// TIA Portal V20 export
// export: Created 2025-12-01T14:57:26.8993515Z, ExportSetting None, DisplayName Totally Integrated Automation Portal, DisplayVersion V20 Update 3, DisplayName TIA Portal Openness, DisplayVersion V20 Update 3, DisplayName TIA Portal Version Control Interface, DisplayVersion V20 Update 3, DisplayName STEP 7 Professional, DisplayVersion V20 Update 3, DisplayName STEP 7 Safety, DisplayVersion V20 Update 2, DisplayName WinCC Basic/Comfort/Advanced, DisplayVersion V20 Update 3, DisplayName WinCC Professional, DisplayVersion V20 Update 3, DisplayName WinCC Unified, DisplayVersion V20 Update 3
FUNCTION "FC606_EventosEnv_Quimarox" : Void   // FC606, LAD
{ S7_Optimized_Access := 'FALSE' }
// stored: AutoNumber false, SetENOAutomatically false
   VAR_INPUT
      NumQuimarox : UInt;
   END_VAR
   VAR_TEMP
      P_Eventos : DWord;
      DBEventos : Word;
      NumDBEventos : UInt;
      MaxBytes : UInt;
      Valor : UDInt;
      NumBytes : UInt;
      Offset : UInt;
      NumVagon : UInt;
      MesaAsociada : UInt;
      MaxNumVagones : UInt;
      EventoAGenerar : UInt;
      Cero : Byte;
      ReturnValor : Int;
      Reserva_Elemento : UInt;
      Reserva_Activa : Bool;
   END_VAR
BEGIN

NETWORK
TITLE = Inicializar
///////////////////////////////////////////////////////////////////////////////////////////
///////////////////////////////////////////////////////////////////////////////////////////
///////////////////////////////////////////////////////////////////////////////////////////
/// Datos del quimarox (Vagon = Peine)
/// ---  Mesa Asociada al Quimarox
/// ---  Maximo Numero de Vagones en el Quimarox

      L     "DB600_ConfigQuimarox".Quimarox[#NumQuimarox].datos_config.Numero_MesaAsociada;
      T     #MesaAsociada;  // Mesa Asociada
      L     "DB600_ConfigQuimarox".Quimarox[#NumQuimarox].datos_config.Numero_vagones;
      T     #MaxNumVagones;  // Numero Maximo De Vagones



NETWORK
TITLE = Comprobacion de Existencia de Eventos en los Vagones
///////////////////////////////////////////////////////////////////////////////////////////
///////////////////////////////////////////////////////////////////////////////////////////
///////////////////////////////////////////////////////////////////////////////////////////
/// Inicio del Recorrido de Vagones Existentes en el Quimarox

      L     1;
      T     #NumVagon;


///////////////////////////////////////////////////////////////////////////////////////////
BucleVagonesQuimarox:NOP   0;
      L     "DB601_PeinesQuimarox".Quimarox[#NumQuimarox].vagon[#NumVagon].EventoAGenerar;
      T     #EventoAGenerar;  // Leer Numero de Evento A Generar

      L     #EventoAGenerar;  // Hay Evento a Generar ?
      L     0;
      <>I;
      JC    GenerarEvento;
      JU    Siguiente_VagonQuimarox;  // Siguiente Vagon


///////////////////////////////////////////////////////////////////////////////////////////
// Continuar Recorriendo los Vagones del Quimarox
Siguiente_VagonQuimarox:NOP   0;
      L     #NumVagon;  // Siguiente Numero de Vagon
      L     1;  // +1
      +I;
      T     #NumVagon;

      L     #NumVagon;  // Es final de los Vagones del Quimarox ?
      L     #MaxNumVagones;
      >I;
      JC    FinalBucleVagonesQuimarox;
      JU    BucleVagonesQuimarox;


///////////////////////////////////////////////////////////////////////////////////////////
///////////////////////////////////////////////////////////////////////////////////////////
///////////////////////////////////////////////////////////////////////////////////////////
/// Final del Recorrido de Vagones existentes en el Quimarox
FinalBucleVagonesQuimarox:NOP   0;
      JU    Final_Funcion;  // Final de la Funcion



NETWORK
TITLE = Inicio de la Generacion del Evento
GenerarEvento:NOP   0;

///////////////////////////////////////////////////////////////////////////////////////////
///////////////////////////////////////////////////////////////////////////////////////////
///////////////////////////////////////////////////////////////////////////////////////////
/// Recoger los Datos del DB a Escribir los Eventos

      L     "JDT1_NDB_EventosEmi";  // Datos del JDT01
      T     #DBEventos;
      T     #NumDBEventos;
      L     "JDT1_MaxBytes";
      T     #MaxBytes;

      SET;
      AN    "DB850_DefinicionMesas".Mesa[#MesaAsociada].ConfigMesa.MesaDeJDT02;
      JC    NoEs_MesaJDT02;  // Es de JDT02 ?


      L     "JDT2_NDB_EventosEmi";  // Datos del JDT02
      T     #DBEventos;
      T     #NumDBEventos;
      L     "JDT2_MaxBytes";
      T     #MaxBytes;

///////////////////////////////////////////////////////////////////////////////////////////
NoEs_MesaJDT02:NOP   0;




NETWORK
TITLE = ---
///////////////////////////////////////////////////////////////////////////////////////////
///////////////////////////////////////////////////////////////////////////////////////////
///////////////////////////////////////////////////////////////////////////////////////////
/// Comprobacion si hay sitio para Formatear el Evento

      L     0;
      T     #NumBytes;  // Inicializo el numero de Bytes
      T     #P_Eventos;  // Inicializo el puntero de Eventos Generados

Inicio_BusquedaFinalEventos:NOP   0;
      OPN   DB [#DBEventos];  // Calcula el tamaño de bytes que hay en el DB
      L     DBB [#P_Eventos];
      L     0;
      ==I;
      JC    Fin_BusquedaFinalEventos;  // Buscamos el final del DB = 0

      OPN   DB [#DBEventos];
      L     DBB [#P_Eventos];
      L     ' ';
      ==I;
      JC    Fin_BusquedaFinalEventos;  // Buscamos el final del DB = ' '

      L     #P_Eventos;  // Incremento de P#1.0
      L     P#1.0;
      +D;
      T     #P_Eventos;

      JU    Inicio_BusquedaFinalEventos;  // Continuar con el siguiente posicion

Fin_BusquedaFinalEventos:NOP   0;
      L     #P_Eventos;  // Sacamos el NumBytes Escritos
      SRD   3;
      T     #NumBytes;

      L     #NumBytes;  // Miramos si hay sitio
      L     #MaxBytes;  // Max. que se pueden emitir, parametro
      >I;
      JC    Final_Funcion;  // No se pueden generar más eventos



NETWORK
TITLE = Distribucion del Evento a Generar
///////////////////////////////////////////////////////////////////////////////////////////
///////////////////////////////////////////////////////////////////////////////////////////
///////////////////////////////////////////////////////////////////////////////////////////
/// Distribucion del Evento a Generar

      L     #EventoAGenerar;
      L     "CTE_InicioEventosQuimarox";
      -I;
      JL    Sin_EventoAGenerar;
      JU    Evento_VagonCargado;  // --- Evento QCAR - Vagon Cargado
      JU    Evento_VagonDesCargado;  // --- Evento QDES - Vagon DesCargado
      JU    Evento_DatosVagon;  // --- Evento QPRE - Datos Existentes en el Vagon
      JU    Evento_DatosVagonReset;  // --- Evento QRST - Datos Existentes en el Vagon en Reset


///////////////////////////////////////////////////////////////////////////////////////////
/// No esta Programado este Evento a Generar
Sin_EventoAGenerar:NOP   0;  // No existe Evento A Generar
      L     0;  // Darlo por tratado
      T     "DB601_PeinesQuimarox".Quimarox[#NumQuimarox].vagon[#NumVagon].EventoAGenerar;
      JU    Siguiente_VagonQuimarox;



NETWORK
TITLE = QCAR (500) - Informa de un Vagon ha sido Cargado con un Movimiento
Evento_VagonCargado:NOP   0;

///////////////////////////////////////////////////////////////////////////////////////////
///////////////////////////////////////////////////////////////////////////////////////////
///////////////////////////////////////////////////////////////////////////////////////////
/// Formatear Evento

      LAR2  #P_Eventos;  // Puntero al DB de Eventos Generados

      TAR2;  // Mirar si es el primer evento de la lista
      L     0;
      ==I;  // Es el primero ?
      JC    NoEsInicio_ListaDeEventos_VagonCargado;

      OPN   DB [#DBEventos];
      L     ',';  // Separador entre eventos ','
      T     DBB [AR2, P#0.0];
      +AR2  P#1.0;

NoEsInicio_ListaDeEventos_VagonCargado:NOP   0;



NETWORK
TITLE = ---- Cuerpo del Evento
///////////////////////////////////////////////////////////////////////////////////////////
///////////////////////////////////////////////////////////////////////////////////////////
///////////////////////////////////////////////////////////////////////////////////////////
/// Cuerpo del Evento
      OPN   DB [#DBEventos];  // DB de Eventos Generados (A Emitir)
      L     '{';  // Inicio de Evento '{'
      T     DBB [AR2, P#0.0];
      +AR2  P#1.0;

      L     'QCAR';  // --- Evento - Movimiento Cargado en el Vagon del Quimarox
      T     DBD [AR2, P#0.0];
      +AR2  P#4.0;


///////////////////////////////////////////////////////////////////////////////////////////
///////////////////////////////////////////////////////////////////////////////////////////
// --- Atributo Numero de Mesa Asociada '[MESA]'
      OPN   DB [#DBEventos];
      L     '[';
      T     DBB [AR2, P#0.0];
      L     'MESA';
      T     DBD [AR2, P#1.0];
      L     ']';
      T     DBB [AR2, P#5.0];
      +AR2  P#6.0;

      L     #MesaAsociada;  // Numero de la Mesa
      L     "CTE_OffsetMesa";
      +I;
      T     #Valor;

// --- Convertir Valor a ASCII
      TAR2;
      SRD   3;
      T     #NumBytes;  // Miro que offset tiene la String

      CALL  "FC893_Obtener_StringDelAtributo"
      ( DB_String := #NumDBEventos,
        OffsetIni := #NumBytes,
        Valor     := #Valor,
        OffsetFin := #Offset
      );  // Llamo a ObtenerString

      L     #Offset;
      SLD   3;
      LAR2;  // Recupero que offset tiene la String
// --- Ya esta convertido el Valor a ASCII


///////////////////////////////////////////////////////////////////////////////////////////
///////////////////////////////////////////////////////////////////////////////////////////
// --- Atributo Numero de Vagon '[VAGO]' J.Zarza: Cambio '[VAGO]' por [PEIN]
      OPN   DB [#DBEventos];
      L     '[';
      T     DBB [AR2, P#0.0];
      L     'PEIN';
      T     DBD [AR2, P#1.0];
      L     ']';
      T     DBB [AR2, P#5.0];
      +AR2  P#6.0;

      L     #NumVagon;  // Numero de Vagon
      T     #Valor;

// --- Convertir Valor a ASCII
      TAR2;
      SRD   3;
      T     #NumBytes;  // Miro que offset tiene la String

      CALL  "FC893_Obtener_StringDelAtributo"
      ( DB_String := #NumDBEventos,
        OffsetIni := #NumBytes,
        Valor     := #Valor,
        OffsetFin := #Offset
      );  // Llamo a ObtenerString

      L     #Offset;
      SLD   3;
      LAR2;  // Recupero que offset tiene la String
// --- Ya esta convertido el Valor a ASCII


///////////////////////////////////////////////////////////////////////////////////////////
///////////////////////////////////////////////////////////////////////////////////////////
// --- Atributo Numero de Movimiento '[MCKY]'
      OPN   DB [#DBEventos];
      L     '[';
      T     DBB [AR2, P#0.0];
      L     'MCKY';
      T     DBD [AR2, P#1.0];
      L     ']';
      T     DBB [AR2, P#5.0];
      +AR2  P#6.0;

      L     "DB601_PeinesQuimarox".Quimarox[#NumQuimarox].vagon[#NumVagon].DatosCarga.Mckey;
      T     #Valor;

// --- Convertir Valor a ASCII
      TAR2;
      SRD   3;
      T     #NumBytes;  // Miro que offset tiene la String

      CALL  "FC893_Obtener_StringDelAtributo"
      ( DB_String := #NumDBEventos,
        OffsetIni := #NumBytes,
        Valor     := #Valor,
        OffsetFin := #Offset
      );  // Llamo a ObtenerString

      L     #Offset;
      SLD   3;
      LAR2;  // Recupero que offset tiene la String
// --- Ya esta convertido el Valor a ASCII


///////////////////////////////////////////////////////////////////////////////////////////
///////////////////////////////////////////////////////////////////////////////////////////
// --- Atributo Numero de Mesa de Carga '[ORIG]'
      OPN   DB [#DBEventos];  // nieves
      L     '[';
      T     DBB [AR2, P#0.0];
      L     'ORIG';
      T     DBD [AR2, P#1.0];
      L     ']';
      T     DBB [AR2, P#5.0];
      +AR2  P#6.0;

      L     "DB601_PeinesQuimarox".Quimarox[#NumQuimarox].vagon[#NumVagon].DatosCarga.MesaOrigen;
      T     #Valor;

// --- Convertir Valor a ASCII
      TAR2;
      SRD   3;
      T     #NumBytes;  // Miro que offset tiene la String

      CALL  "FC893_Obtener_StringDelAtributo"
      ( DB_String := #NumDBEventos,
        OffsetIni := #NumBytes,
        Valor     := #Valor,
        OffsetFin := #Offset
      );  // Llamo a ObtenerString

      L     #Offset;
      SLD   3;
      LAR2;  // Recupero que offset tiene la String
// --- Ya esta convertido el Valor a ASCII


///////////////////////////////////////////////////////////////////////////////////////////
///////////////////////////////////////////////////////////////////////////////////////////
// --- Atributo Numero de Mesa de DesCarga '[DEST]'
      OPN   DB [#DBEventos];
      L     '[';
      T     DBB [AR2, P#0.0];
      L     'DEST';
      T     DBD [AR2, P#1.0];
      L     ']';
      T     DBB [AR2, P#5.0];
      +AR2  P#6.0;

      L     "DB601_PeinesQuimarox".Quimarox[#NumQuimarox].vagon[#NumVagon].DatosCarga.MesaDestino;
      T     #Valor;

// --- Convertir Valor a ASCII
      TAR2;
      SRD   3;
      T     #NumBytes;  // Miro que offset tiene la String

      CALL  "FC893_Obtener_StringDelAtributo"
      ( DB_String := #NumDBEventos,
        OffsetIni := #NumBytes,
        Valor     := #Valor,
        OffsetFin := #Offset
      );  // Llamo a ObtenerString

      L     #Offset;
      SLD   3;
      LAR2;  // Recupero que offset tiene la String
// --- Ya esta convertido el Valor a ASCII


///////////////////////////////////////////////////////////////////////////////////////////
///////////////////////////////////////////////////////////////////////////////////////////
// --- Atributo Etiqueta '[SSCC]'

      SET;  // --- Comprobar si tiene que ir en el Evento
      AN    "DB600_ConfigQuimarox".Quimarox[#NumQuimarox].datos_config.ConfigEvento.SSCC;
      JC    NoConfiguradoAtributo_SCCC_EventoVagonCargado;


///////////////////////////////////////////////////////////////////////////////////////////
      OPN   DB [#DBEventos];
      L     '[';
      T     DBB [AR2, P#0.0];
      L     'SSCC';
      T     DBD [AR2, P#1.0];
      L     ']';
      T     DBB [AR2, P#5.0];
      +AR2  P#6.0;

      L     "DB601_PeinesQuimarox".Quimarox[#NumQuimarox].vagon[#NumVagon].DatosCarga.EtiquetaRouter;
      T     #Valor;

// --- Convertir Valor a ASCII
      TAR2;
      SRD   3;
      T     #NumBytes;  // Miro que offset tiene la String

      CALL  "FC893_Obtener_StringDelAtributo"
      ( DB_String := #NumDBEventos,
        OffsetIni := #NumBytes,
        Valor     := #Valor,
        OffsetFin := #Offset
      );  // Llamo a ObtenerString

      L     #Offset;
      SLD   3;
      LAR2;  // Recupero que offset tiene la String
// --- Ya esta convertido el Valor a ASCII


///////////////////////////////////////////////////////////////////////////////////////////
NoConfiguradoAtributo_SCCC_EventoVagonCargado:NOP   0;



NETWORK
TITLE = ---- Final del Evento
///////////////////////////////////////////////////////////////////////////////////////////
///////////////////////////////////////////////////////////////////////////////////////////
/// Final del Evento

      OPN   DB [#DBEventos];  // DB de Eventos Generados (A Emitir)
      L     '}';  // --- Fin de Evento '}'
      T     DBB [AR2, P#0.0];
      +AR2  P#1.0;


///////////////////////////////////////////////////////////////////////////////////////////
///////////////////////////////////////////////////////////////////////////////////////////
/// Final del formateo del evento

      L     0;  // Darlo por tratado
      T     "DB601_PeinesQuimarox".Quimarox[#NumQuimarox].vagon[#NumVagon].EventoAGenerar;

      JU    Siguiente_VagonQuimarox;  // Siguiente Vagon



NETWORK
TITLE = QDES (501) - Informa de una Vagon ha sido DesCargado de un Movimiento
Evento_VagonDesCargado:NOP   0;

///////////////////////////////////////////////////////////////////////////////////////////
///////////////////////////////////////////////////////////////////////////////////////////
///////////////////////////////////////////////////////////////////////////////////////////
/// Formatear Evento

      LAR2  #P_Eventos;  // Puntero al DB de Eventos Generados

      TAR2;  // Mirar si es el primer evento de la lista
      L     0;
      ==I;  // Es el primero ?
      JC    NoEsInicio_ListaDeEventos_VagonDesCargado;

      OPN   DB [#DBEventos];
      L     ',';  // Separador entre eventos ','
      T     DBB [AR2, P#0.0];
      +AR2  P#1.0;

NoEsInicio_ListaDeEventos_VagonDesCargado:NOP   0;



NETWORK
TITLE = ---- Cuerpo del Evento.
///////////////////////////////////////////////////////////////////////////////////////////
///////////////////////////////////////////////////////////////////////////////////////////
///////////////////////////////////////////////////////////////////////////////////////////
/// Cuerpo del Evento
      OPN   DB [#DBEventos];  // DB de Eventos Generados (A Emitir)
      L     '{';  // Inicio de Evento '{'
      T     DBB [AR2, P#0.0];
      +AR2  P#1.0;

      L     'QDES';  // --- Evento - Movimiento DesCargado del Vagon del Quimarox
      T     DBD [AR2, P#0.0];
      +AR2  P#4.0;


///////////////////////////////////////////////////////////////////////////////////////////
///////////////////////////////////////////////////////////////////////////////////////////
// --- Atributo Numero de Mesa Asociada '[MESA]'
      OPN   DB [#DBEventos];  // DB de Eventos Generados (A Emitir)
      L     '[';
      T     DBB [AR2, P#0.0];
      L     'MESA';
      T     DBD [AR2, P#1.0];
      L     ']';
      T     DBB [AR2, P#5.0];
      +AR2  P#6.0;

      L     #MesaAsociada;  // Numero de la Mesa
      L     "CTE_OffsetMesa";
      +I;
      T     #Valor;

// --- Convertir Valor a ASCII
      TAR2;
      SRD   3;
      T     #NumBytes;  // Miro que offset tiene la String

      CALL  "FC893_Obtener_StringDelAtributo"
      ( DB_String := #NumDBEventos,
        OffsetIni := #NumBytes,
        Valor     := #Valor,
        OffsetFin := #Offset
      );  // Llamo a ObtenerString

      L     #Offset;
      SLD   3;
      LAR2;  // Recupero que offset tiene la String
// --- Ya esta convertido el Valor a ASCII


///////////////////////////////////////////////////////////////////////////////////////////
///////////////////////////////////////////////////////////////////////////////////////////
// --- Atributo Numero de Vagon '[VAGO]' J.Zarza: Cambio '[VAGO]' por [PEIN]
      OPN   DB [#DBEventos];  // DB de Eventos Generados (A Emitir)
      L     '[';
      T     DBB [AR2, P#0.0];
      L     'PEIN';
      T     DBD [AR2, P#1.0];
      L     ']';
      T     DBB [AR2, P#5.0];
      +AR2  P#6.0;

      L     #NumVagon;  // Numero de Vagon
      T     #Valor;

// --- Convertir Valor a ASCII
      TAR2;
      SRD   3;
      T     #NumBytes;  // Miro que offset tiene la String

      CALL  "FC893_Obtener_StringDelAtributo"
      ( DB_String := #NumDBEventos,
        OffsetIni := #NumBytes,
        Valor     := #Valor,
        OffsetFin := #Offset
      );  // Llamo a ObtenerString

      L     #Offset;
      SLD   3;
      LAR2;  // Recupero que offset tiene la String
// --- Ya esta convertido el Valor a ASCII


///////////////////////////////////////////////////////////////////////////////////////////
///////////////////////////////////////////////////////////////////////////////////////////
// --- Atributo Numero de Movimiento '[MCKY]'
      OPN   DB [#DBEventos];  // DB de Eventos Generados (A Emitir)
      L     '[';
      T     DBB [AR2, P#0.0];
      L     'MCKY';
      T     DBD [AR2, P#1.0];
      L     ']';
      T     DBB [AR2, P#5.0];
      +AR2  P#6.0;

      L     "DB601_PeinesQuimarox".Quimarox[#NumQuimarox].vagon[#NumVagon].DatosCarga.Mckey;
      T     #Valor;

// --- Convertir Valor a ASCII
      TAR2;
      SRD   3;
      T     #NumBytes;  // Miro que offset tiene la String

      CALL  "FC893_Obtener_StringDelAtributo"
      ( DB_String := #NumDBEventos,
        OffsetIni := #NumBytes,
        Valor     := #Valor,
        OffsetFin := #Offset
      );  // Llamo a ObtenerString

      L     #Offset;
      SLD   3;
      LAR2;  // Recupero que offset tiene la String
// --- Ya esta convertido el Valor a ASCII


///////////////////////////////////////////////////////////////////////////////////////////
///////////////////////////////////////////////////////////////////////////////////////////
// --- Atributo Numero de Mesa de DesCarga '[DEST]'
      OPN   DB [#DBEventos];
      L     '[';
      T     DBB [AR2, P#0.0];
      L     'ORIG';
      T     DBD [AR2, P#1.0];
      L     ']';
      T     DBB [AR2, P#5.0];
      +AR2  P#6.0;

      L     "DB601_PeinesQuimarox".Quimarox[#NumQuimarox].vagon[#NumVagon].DatosCarga.MesaOrigen;
      T     #Valor;

// --- Convertir Valor a ASCII
      TAR2;
      SRD   3;
      T     #NumBytes;  // Miro que offset tiene la String

      CALL  "FC893_Obtener_StringDelAtributo"
      ( DB_String := #NumDBEventos,
        OffsetIni := #NumBytes,
        Valor     := #Valor,
        OffsetFin := #Offset
      );  // Llamo a ObtenerString

      L     #Offset;
      SLD   3;
      LAR2;  // Recupero que offset tiene la String
// --- Ya esta convertido el Valor a ASCII


///////////////////////////////////////////////////////////////////////////////////////////
///////////////////////////////////////////////////////////////////////////////////////////
// --- Atributo Numero de Mesa de DesCarga '[DEST]'
      OPN   DB [#DBEventos];
      L     '[';
      T     DBB [AR2, P#0.0];
      L     'DEST';
      T     DBD [AR2, P#1.0];
      L     ']';
      T     DBB [AR2, P#5.0];
      +AR2  P#6.0;

      L     "DB601_PeinesQuimarox".Quimarox[#NumQuimarox].vagon[#NumVagon].DatosCarga.MesaDestino;
      T     #Valor;

// --- Convertir Valor a ASCII
      TAR2;
      SRD   3;
      T     #NumBytes;  // Miro que offset tiene la String

      CALL  "FC893_Obtener_StringDelAtributo"
      ( DB_String := #NumDBEventos,
        OffsetIni := #NumBytes,
        Valor     := #Valor,
        OffsetFin := #Offset
      );  // Llamo a ObtenerString

      L     #Offset;
      SLD   3;
      LAR2;  // Recupero que offset tiene la String
// --- Ya esta convertido el Valor a ASCII


///////////////////////////////////////////////////////////////////////////////////////////

///////////////////////////////////////////////////////////////////////////////////////////
// --- Atributo Numero de Mesa de DesCarga '[DESC]'
      OPN   DB [#DBEventos];
      L     '[';
      T     DBB [AR2, P#0.0];
      L     'DESC';
      T     DBD [AR2, P#1.0];
      L     ']';
      T     DBB [AR2, P#5.0];
      +AR2  P#6.0;

      L     "DB601_PeinesQuimarox".Quimarox[#NumQuimarox].vagon[#NumVagon].Mesa_descarga;
      T     #Valor;

// --- Convertir Valor a ASCII
      TAR2;
      SRD   3;
      T     #NumBytes;  // Miro que offset tiene la String

      CALL  "FC893_Obtener_StringDelAtributo"
      ( DB_String := #NumDBEventos,
        OffsetIni := #NumBytes,
        Valor     := #Valor,
        OffsetFin := #Offset
      );  // Llamo a ObtenerString

      L     #Offset;
      SLD   3;
      LAR2;  // Recupero que offset tiene la String
// --- Ya esta convertido el Valor a ASCII


///////////////////////////////////////////////////////////////////////////////////////////
///////////////////////////////////////////////////////////////////////////////////////////
// --- Atributo Etiqueta '[SSCC]'

      SET;  // --- Comprobar si tiene que ir en el Evento
      AN    "DB600_ConfigQuimarox".Quimarox[#NumQuimarox].datos_config.ConfigEvento.SSCC;
      JC    NoConfiguradoAtributo_SCCC_EventoVagonDesCargado;


///////////////////////////////////////////////////////////////////////////////////////////
      OPN   DB [#DBEventos];
      L     '[';
      T     DBB [AR2, P#0.0];
      L     'SSCC';
      T     DBD [AR2, P#1.0];
      L     ']';
      T     DBB [AR2, P#5.0];
      +AR2  P#6.0;

      L     "DB601_PeinesQuimarox".Quimarox[#NumQuimarox].vagon[#NumVagon].DatosCarga.EtiquetaRouter;
      T     #Valor;

// --- Convertir Valor a ASCII
      TAR2;
      SRD   3;
      T     #NumBytes;  // Miro que offset tiene la String

      CALL  "FC893_Obtener_StringDelAtributo"
      ( DB_String := #NumDBEventos,
        OffsetIni := #NumBytes,
        Valor     := #Valor,
        OffsetFin := #Offset
      );  // Llamo a ObtenerString

      L     #Offset;
      SLD   3;
      LAR2;  // Recupero que offset tiene la String
// --- Ya esta convertido el Valor a ASCII


///////////////////////////////////////////////////////////////////////////////////////////
NoConfiguradoAtributo_SCCC_EventoVagonDesCargado:NOP   0;



NETWORK
TITLE = ---- Final del Evento
///////////////////////////////////////////////////////////////////////////////////////////
///////////////////////////////////////////////////////////////////////////////////////////
/// Final del Evento

      OPN   DB [#DBEventos];  // DB de Eventos Generados (A Emitir)
      L     '}';  // --- Fin de Evento '}'
      T     DBB [AR2, P#0.0];
      +AR2  P#1.0;


///////////////////////////////////////////////////////////////////////////////////////////
///////////////////////////////////////////////////////////////////////////////////////////
/// Final del formateo del evento
// --- Guardar Reserva
      SET;
      A     "DB601_PeinesQuimarox".Quimarox[#NumQuimarox].vagon[#NumVagon].vagon_reservado_carga;
      =     #Reserva_Activa;

      L     "DB601_PeinesQuimarox".Quimarox[#NumQuimarox].vagon[#NumVagon].punto_entrada_carga;
      T     #Reserva_Elemento;

// --- Borrado de datos del Vagon
      L     0;
      T     #Cero;
      CALL  FILL
      ( BVAL    := #Cero,
        RET_VAL := #ReturnValor,
        BLK     := "DB601_PeinesQuimarox".Quimarox[#NumQuimarox].vagon[#NumVagon]
      );

// --- Recuperar Reserva
      SET;
      A     #Reserva_Activa;
      =     "DB601_PeinesQuimarox".Quimarox[#NumQuimarox].vagon[#NumVagon].vagon_reservado_carga;

      L     #Reserva_Elemento;
      T     "DB601_PeinesQuimarox".Quimarox[#NumQuimarox].vagon[#NumVagon].punto_entrada_carga;

      JU    Siguiente_VagonQuimarox;  // Siguiente Vagon



NETWORK
TITLE = QPRE (502) - Informa de Presencia de Carga en un Vagon
Evento_DatosVagon:NOP   0;

///////////////////////////////////////////////////////////////////////////////////////////
///////////////////////////////////////////////////////////////////////////////////////////
///////////////////////////////////////////////////////////////////////////////////////////
/// Formatear Evento

      LAR2  #P_Eventos;  // Puntero al DB de Eventos Generados

      TAR2;  // Mirar si es el primer evento de la lista
      L     0;
      ==I;  // Es el primero ?
      JC    NoEsInicio_ListaDeEventos_DatosVagon;

      OPN   DB [#DBEventos];
      L     ',';  // Separador entre eventos ','
      T     DBB [AR2, P#0.0];
      +AR2  P#1.0;

NoEsInicio_ListaDeEventos_DatosVagon:NOP   0;



NETWORK
TITLE = ---- Cuerpo del Evento.
///////////////////////////////////////////////////////////////////////////////////////////
///////////////////////////////////////////////////////////////////////////////////////////
///////////////////////////////////////////////////////////////////////////////////////////
/// Cuerpo del Evento
      OPN   DB [#DBEventos];  // DB de Eventos Generados (A Emitir)
      L     '{';  // Inicio de Evento '{'
      T     DBB [AR2, P#0.0];
      +AR2  P#1.0;

      L     'QPRE';  // --- Evento - Informa de la Datos del Vagon del Quimarox (Solo Carga)
      T     DBD [AR2, P#0.0];
      +AR2  P#4.0;


///////////////////////////////////////////////////////////////////////////////////////////
///////////////////////////////////////////////////////////////////////////////////////////
// --- Atributo Numero de Mesa Asociada '[MESA]'
      OPN   DB [#DBEventos];
      L     '[';
      T     DBB [AR2, P#0.0];
      L     'MESA';
      T     DBD [AR2, P#1.0];
      L     ']';
      T     DBB [AR2, P#5.0];
      +AR2  P#6.0;

      L     #MesaAsociada;  // Numero de la Mesa
      L     "CTE_OffsetMesa";
      +I;
      T     #Valor;

// --- Convertir Valor a ASCII
      TAR2;
      SRD   3;
      T     #NumBytes;  // Miro que offset tiene la String

      CALL  "FC893_Obtener_StringDelAtributo"
      ( DB_String := #NumDBEventos,
        OffsetIni := #NumBytes,
        Valor     := #Valor,
        OffsetFin := #Offset
      );  // Llamo a ObtenerString

      L     #Offset;
      SLD   3;
      LAR2;  // Recupero que offset tiene la String
// --- Ya esta convertido el Valor a ASCII


///////////////////////////////////////////////////////////////////////////////////////////
///////////////////////////////////////////////////////////////////////////////////////////
// --- Atributo Numero de Vagon '[VAGO]' J.Z. Cambio atributo de VAGO a PEIN
      OPN   DB [#DBEventos];
      L     '[';
      T     DBB [AR2, P#0.0];
      L     'PEIN';
      T     DBD [AR2, P#1.0];
      L     ']';
      T     DBB [AR2, P#5.0];
      +AR2  P#6.0;

      L     #NumVagon;  // Numero de Vagon
      T     #Valor;

// --- Convertir Valor a ASCII
      TAR2;
      SRD   3;
      T     #NumBytes;  // Miro que offset tiene la String

      CALL  "FC893_Obtener_StringDelAtributo"
      ( DB_String := #NumDBEventos,
        OffsetIni := #NumBytes,
        Valor     := #Valor,
        OffsetFin := #Offset
      );  // Llamo a ObtenerString

      L     #Offset;
      SLD   3;
      LAR2;  // Recupero que offset tiene la String
// --- Ya esta convertido el Valor a ASCII


///////////////////////////////////////////////////////////////////////////////////////////
///////////////////////////////////////////////////////////////////////////////////////////
// --- Atributo Numero de Movimiento '[MCKY]'
      OPN   DB [#DBEventos];
      L     '[';
      T     DBB [AR2, P#0.0];
      L     'MCKY';
      T     DBD [AR2, P#1.0];
      L     ']';
      T     DBB [AR2, P#5.0];
      +AR2  P#6.0;

      L     "DB601_PeinesQuimarox".Quimarox[#NumQuimarox].vagon[#NumVagon].DatosCarga.Mckey;
      T     #Valor;

// --- Convertir Valor a ASCII
      TAR2;
      SRD   3;
      T     #NumBytes;  // Miro que offset tiene la String

      CALL  "FC893_Obtener_StringDelAtributo"
      ( DB_String := #NumDBEventos,
        OffsetIni := #NumBytes,
        Valor     := #Valor,
        OffsetFin := #Offset
      );  // Llamo a ObtenerString

      L     #Offset;
      SLD   3;
      LAR2;  // Recupero que offset tiene la String
// --- Ya esta convertido el Valor a ASCII


///////////////////////////////////////////////////////////////////////////////////////////
///////////////////////////////////////////////////////////////////////////////////////////
// --- Atributo Numero de Mesa de DesCarga '[DESC]'
      OPN   DB [#DBEventos];
      L     '[';
      T     DBB [AR2, P#0.0];
      L     'ORIG';
      T     DBD [AR2, P#1.0];
      L     ']';
      T     DBB [AR2, P#5.0];
      +AR2  P#6.0;

      L     "DB601_PeinesQuimarox".Quimarox[#NumQuimarox].vagon[#NumVagon].DatosCarga.MesaOrigen;
      T     #Valor;

// --- Convertir Valor a ASCII
      TAR2;
      SRD   3;
      T     #NumBytes;  // Miro que offset tiene la String

      CALL  "FC893_Obtener_StringDelAtributo"
      ( DB_String := #NumDBEventos,
        OffsetIni := #NumBytes,
        Valor     := #Valor,
        OffsetFin := #Offset
      );

      L     #Offset;
      SLD   3;
      LAR2;  // Recupero que offset tiene la String
// --- Ya esta convertido el Valor a ASCII


///////////////////////////////////////////////////////////////////////////////////////////
///////////////////////////////////////////////////////////////////////////////////////////
// --- Atributo Numero de Mesa de DesCarga '[DESC]'
      OPN   DB [#DBEventos];
      L     '[';
      T     DBB [AR2, P#0.0];
      L     'DEST';
      T     DBD [AR2, P#1.0];
      L     ']';
      T     DBB [AR2, P#5.0];
      +AR2  P#6.0;

      L     "DB601_PeinesQuimarox".Quimarox[#NumQuimarox].vagon[#NumVagon].DatosCarga.MesaDestino;
      T     #Valor;

// --- Convertir Valor a ASCII
      TAR2;
      SRD   3;
      T     #NumBytes;  // Miro que offset tiene la String

      CALL  "FC893_Obtener_StringDelAtributo"
      ( DB_String := #NumDBEventos,
        OffsetIni := #NumBytes,
        Valor     := #Valor,
        OffsetFin := #Offset
      );  // Llamo a ObtenerString

      L     #Offset;
      SLD   3;
      LAR2;  // Recupero que offset tiene la String
// --- Ya esta convertido el Valor a ASCII


///////////////////////////////////////////////////////////////////////////////////////////
///////////////////////////////////////////////////////////////////////////////////////////
// --- Atributo Etiqueta '[SSCC]'
      SET;  // --- Comprobar si tiene que ir en el Evento
      AN    "DB600_ConfigQuimarox".Quimarox[#NumQuimarox].datos_config.ConfigEvento.SSCC;
      JC    NoConfiguradoAtributo_SCCC_EventoDatosVagon;


///////////////////////////////////////////////////////////////////////////////////////////
      OPN   DB [#DBEventos];
      L     '[';
      T     DBB [AR2, P#0.0];
      L     'SSCC';
      T     DBD [AR2, P#1.0];
      L     ']';
      T     DBB [AR2, P#5.0];
      +AR2  P#6.0;

      L     "DB601_PeinesQuimarox".Quimarox[#NumQuimarox].vagon[#NumVagon].DatosCarga.EtiquetaRouter;
      T     #Valor;

// --- Convertir Valor a ASCII
      TAR2;
      SRD   3;
      T     #NumBytes;  // Miro que offset tiene la String

      CALL  "FC893_Obtener_StringDelAtributo"
      ( DB_String := #NumDBEventos,
        OffsetIni := #NumBytes,
        Valor     := #Valor,
        OffsetFin := #Offset
      );  // Llamo a ObtenerString

      L     #Offset;
      SLD   3;
      LAR2;  // Recupero que offset tiene la String
// --- Ya esta convertido el Valor a ASCII


///////////////////////////////////////////////////////////////////////////////////////////
NoConfiguradoAtributo_SCCC_EventoDatosVagon:NOP   0;



NETWORK
TITLE = ---- Final del Evento
///////////////////////////////////////////////////////////////////////////////////////////
///////////////////////////////////////////////////////////////////////////////////////////
/// Final del Evento

      OPN   DB [#DBEventos];  // DB de Eventos Generados (A Emitir)
      L     '}';  // --- Fin de Evento '}'
      T     DBB [AR2, P#0.0];
      +AR2  P#1.0;


///////////////////////////////////////////////////////////////////////////////////////////
///////////////////////////////////////////////////////////////////////////////////////////
/// Final del formateo del evento

      L     0;  // Darlo por tratado
      T     "DB601_PeinesQuimarox".Quimarox[#NumQuimarox].vagon[#NumVagon].EventoAGenerar;

      JU    Siguiente_VagonQuimarox;  // Siguiente Vagon




NETWORK
TITLE = QRST (503) - Informa de Presencia de Carga en un Vagon en Reset
Evento_DatosVagonReset:NOP   0;

///////////////////////////////////////////////////////////////////////////////////////////
///////////////////////////////////////////////////////////////////////////////////////////
///////////////////////////////////////////////////////////////////////////////////////////
/// Formatear Evento

      LAR2  #P_Eventos;  // Puntero al DB de Eventos Generados

      TAR2;  // Mirar si es el primer evento de la lista
      L     0;
      ==I;  // Es el primero ?
      JC    NoEsInicio_ListaDeEventos_DatosVagonReset;

      OPN   DB [#DBEventos];
      L     ',';  // Separador entre eventos ','
      T     DBB [AR2, P#0.0];
      +AR2  P#1.0;

NoEsInicio_ListaDeEventos_DatosVagonReset:NOP   0;



NETWORK
TITLE = ---- Cuerpo del Evento
///////////////////////////////////////////////////////////////////////////////////////////
///////////////////////////////////////////////////////////////////////////////////////////
///////////////////////////////////////////////////////////////////////////////////////////
/// Cuerpo del Evento
      OPN   DB [#DBEventos];  // DB de Eventos Generados (A Emitir)
      L     '{';  // Inicio de Evento '{'
      T     DBB [AR2, P#0.0];
      +AR2  P#1.0;

      L     'QRST';  // --- Evento - Informa de la Datos del Vagon del Quimarox (Solo Carga)
      T     DBD [AR2, P#0.0];
      +AR2  P#4.0;


///////////////////////////////////////////////////////////////////////////////////////////
///////////////////////////////////////////////////////////////////////////////////////////
// --- Atributo Numero de Mesa Asociada '[MESA]'
      OPN   DB [#DBEventos];
      L     '[';
      T     DBB [AR2, P#0.0];
      L     'MESA';
      T     DBD [AR2, P#1.0];
      L     ']';
      T     DBB [AR2, P#5.0];
      +AR2  P#6.0;

      L     #MesaAsociada;  // Numero de la Mesa
      L     "CTE_OffsetMesa";
      +I;
      T     #Valor;

// --- Convertir Valor a ASCII
      TAR2;
      SRD   3;
      T     #NumBytes;  // Miro que offset tiene la String

      CALL  "FC893_Obtener_StringDelAtributo"
      ( DB_String := #NumDBEventos,
        OffsetIni := #NumBytes,
        Valor     := #Valor,
        OffsetFin := #Offset
      );  // Llamo a ObtenerString

      L     #Offset;
      SLD   3;
      LAR2;  // Recupero que offset tiene la String
// --- Ya esta convertido el Valor a ASCII


///////////////////////////////////////////////////////////////////////////////////////////
///////////////////////////////////////////////////////////////////////////////////////////
// --- Atributo Numero de Vagon '[VAGO]' J.Zarza Cambio atributo de VAGO a PEIN
      OPN   DB [#DBEventos];
      L     '[';
      T     DBB [AR2, P#0.0];
      L     'PEIN';
      T     DBD [AR2, P#1.0];
      L     ']';
      T     DBB [AR2, P#5.0];
      +AR2  P#6.0;

      L     #NumVagon;  // Numero de Vagon
      T     #Valor;

// --- Convertir Valor a ASCII
      TAR2;
      SRD   3;
      T     #NumBytes;  // Miro que offset tiene la String

      CALL  "FC893_Obtener_StringDelAtributo"
      ( DB_String := #NumDBEventos,
        OffsetIni := #NumBytes,
        Valor     := #Valor,
        OffsetFin := #Offset
      );  // Llamo a ObtenerString

      L     #Offset;
      SLD   3;
      LAR2;  // Recupero que offset tiene la String
// --- Ya esta convertido el Valor a ASCII


///////////////////////////////////////////////////////////////////////////////////////////
///////////////////////////////////////////////////////////////////////////////////////////
// --- Atributo Numero de Movimiento '[MCKY]'
      OPN   DB [#DBEventos];
      L     '[';
      T     DBB [AR2, P#0.0];
      L     'MCKY';
      T     DBD [AR2, P#1.0];
      L     ']';
      T     DBB [AR2, P#5.0];
      +AR2  P#6.0;

      L     "DB601_PeinesQuimarox".Quimarox[#NumQuimarox].vagon[#NumVagon].DatosCarga.Mckey;
      T     #Valor;

// --- Convertir Valor a ASCII
      TAR2;
      SRD   3;
      T     #NumBytes;  // Miro que offset tiene la String

      CALL  "FC893_Obtener_StringDelAtributo"
      ( DB_String := #NumDBEventos,
        OffsetIni := #NumBytes,
        Valor     := #Valor,
        OffsetFin := #Offset
      );  // Llamo a ObtenerString

      L     #Offset;
      SLD   3;
      LAR2;  // Recupero que offset tiene la String
// --- Ya esta convertido el Valor a ASCII

///////////////////////////////////////////////////////////////////////////////////////////
///////////////////////////////////////////////////////////////////////////////////////////
// --- Atributo Numero de Mesa de DesCarga '[DESC]'
      OPN   DB [#DBEventos];
      L     '[';
      T     DBB [AR2, P#0.0];
      L     'ORIG';
      T     DBD [AR2, P#1.0];
      L     ']';
      T     DBB [AR2, P#5.0];
      +AR2  P#6.0;

      L     "DB601_PeinesQuimarox".Quimarox[#NumQuimarox].vagon[#NumVagon].DatosCarga.MesaOrigen;
      T     #Valor;

// --- Convertir Valor a ASCII
      TAR2;
      SRD   3;
      T     #NumBytes;  // Miro que offset tiene la String

      CALL  "FC893_Obtener_StringDelAtributo"
      ( DB_String := #NumDBEventos,
        OffsetIni := #NumBytes,
        Valor     := #Valor,
        OffsetFin := #Offset
      );  // Llamo a ObtenerString

      L     #Offset;
      SLD   3;
      LAR2;  // Recupero que offset tiene la String
// --- Ya esta convertido el Valor a ASCII


///////////////////////////////////////////////////////////////////////////////////////////
///////////////////////////////////////////////////////////////////////////////////////////
// --- Atributo Numero de Mesa de DesCarga '[DESC]'
      OPN   DB [#DBEventos];
      L     '[';
      T     DBB [AR2, P#0.0];
      L     'DEST';
      T     DBD [AR2, P#1.0];
      L     ']';
      T     DBB [AR2, P#5.0];
      +AR2  P#6.0;

      L     "DB601_PeinesQuimarox".Quimarox[#NumQuimarox].vagon[#NumVagon].DatosCarga.MesaDestino;
      T     #Valor;

// --- Convertir Valor a ASCII
      TAR2;
      SRD   3;
      T     #NumBytes;  // Miro que offset tiene la String

      CALL  "FC893_Obtener_StringDelAtributo"
      ( DB_String := #NumDBEventos,
        OffsetIni := #NumBytes,
        Valor     := #Valor,
        OffsetFin := #Offset
      );  // Llamo a ObtenerString

      L     #Offset;
      SLD   3;
      LAR2;  // Recupero que offset tiene la String
// --- Ya esta convertido el Valor a ASCII


///////////////////////////////////////////////////////////////////////////////////////////
///////////////////////////////////////////////////////////////////////////////////////////
// --- Atributo Etiqueta '[SSCC]'
      SET;  // --- Comprobar si tiene que ir en el Evento
      AN    "DB600_ConfigQuimarox".Quimarox[#NumQuimarox].datos_config.ConfigEvento.SSCC;
      JC    NoConfiguradoAtributo_SCCC_EventoDatosVagonReset;


///////////////////////////////////////////////////////////////////////////////////////////
      OPN   DB [#DBEventos];
      L     '[';
      T     DBB [AR2, P#0.0];
      L     'SSCC';
      T     DBD [AR2, P#1.0];
      L     ']';
      T     DBB [AR2, P#5.0];
      +AR2  P#6.0;

      L     "DB601_PeinesQuimarox".Quimarox[#NumQuimarox].vagon[#NumVagon].DatosCarga.EtiquetaRouter;
      T     #Valor;

// --- Convertir Valor a ASCII
      TAR2;
      SRD   3;
      T     #NumBytes;  // Miro que offset tiene la String

      CALL  "FC893_Obtener_StringDelAtributo"
      ( DB_String := #NumDBEventos,
        OffsetIni := #NumBytes,
        Valor     := #Valor,
        OffsetFin := #Offset
      );  // Llamo a ObtenerString

      L     #Offset;
      SLD   3;
      LAR2;  // Recupero que offset tiene la String
// --- Ya esta convertido el Valor a ASCII


///////////////////////////////////////////////////////////////////////////////////////////
NoConfiguradoAtributo_SCCC_EventoDatosVagonReset:NOP   0;



NETWORK
TITLE = ---- Final del Evento
///////////////////////////////////////////////////////////////////////////////////////////
///////////////////////////////////////////////////////////////////////////////////////////
/// Final del Evento

      OPN   DB [#DBEventos];  // DB de Eventos Generados (A Emitir)
      L     '}';  // --- Fin de Evento '}'
      T     DBB [AR2, P#0.0];
      +AR2  P#1.0;


///////////////////////////////////////////////////////////////////////////////////////////
///////////////////////////////////////////////////////////////////////////////////////////
/// Final del formateo del evento

      L     0;  // Darlo por tratado
      T     "DB601_PeinesQuimarox".Quimarox[#NumQuimarox].vagon[#NumVagon].EventoAGenerar;

      L     0;  // Brorardo de Peine
      T     #Cero;
      CALL  FILL
      ( BVAL    := #Cero,
        RET_VAL := #ReturnValor,
        BLK     := "DB601_PeinesQuimarox".Quimarox[#NumQuimarox].vagon[#NumVagon]
      );

      JU    Siguiente_VagonQuimarox;  // Siguiente Vagon




NETWORK
TITLE = Final de la Funcion
///////////////////////////////////////////////////////////////////////////////////////////
///////////////////////////////////////////////////////////////////////////////////////////
///////////////////////////////////////////////////////////////////////////////////////////
/// Se ha acabo la funcion
Final_Funcion:NOP   0;


END_FUNCTION
